// TIA Portal V19 export
TYPE "_IOL_VMrdParInterface"
   STRUCT
      ia : Struct   // Parameters ANY Pointer
         dbno : Int := 28;   // DB Number
         sta : Int;   // Starting Address (Byte offset)
         al : Int;   // Area Length in bytes
      END_STRUCT;
      dataStore : Struct   // Parameters ANY Pointer
         dbno : Int := 28;   // DB Number
         sta : Int;   // Starting Address (Byte offset)
         al : Int;   // Area Length in bytes
      END_STRUCT;
   END_STRUCT;
END_TYPE
